// TIA Portal V17 export
// export: Created 2024-09-02T12:50:41.1699266Z, ExportSetting WithDefaults, DisplayName Totally Integrated Automation Portal, DisplayVersion V17, DisplayName TIA Portal Openness, DisplayVersion V17, DisplayName TIA Portal Version Control Interface, DisplayVersion V17, DisplayName STEP 7 Professional, DisplayVersion V17, DisplayName STEP 7 Safety, DisplayVersion V17, DisplayName WinCC Professional, DisplayVersion V17
TYPE "Aveva_Specyfication_General_Info"
// stored: IsFailsafeCompliant false
   STRUCT
      PalletID { ExternalWritable := 'False'} : String[25];   // Unique Pallet ID/Product ID
      TimeStamp { ExternalWritable := 'False'} : LDT;
      iSynchro : Int;   // Synchronization word between PLC Concentrator/PLC Workstation
      iDefault : String;   // Default Word
      ProductStatus : Int;   // Product status of the previous Workstation 1 = OK, 2 = NOK, 3 = empty pallet
   END_STRUCT;
END_TYPE
